RoboDK station: New Station (1).rdk

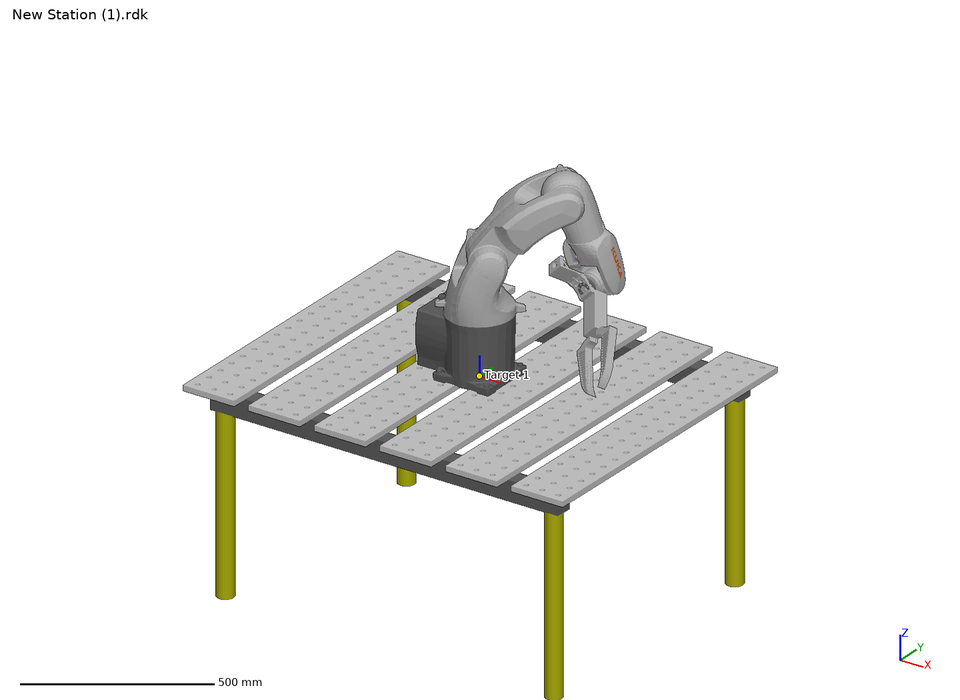
[picture v0: the station drawn from its stored meshes, robots at their saved joint values, targets as dots, program paths as lines]
Station New Station (1). Poses are relative to the parent item; angles as X-Y-Z fixed-axis rotations.
Station parameters (name, value as stored): DO_NAME, 1, IO_2, 0, IO_1, 1
  - object Table at (0, 1063.9, 0) mm, size 1193.8 x 965.2 x 609.6 mm, geometry from welding_table.sld
  - frame KUKA KR 3 R540 Base at (0, 1061.83, 0) mm
    - robot KUKA KR 3 R540: 6 axes, payload 3 kg, reach 541 mm, repeatability 0.02 mm, weight 26 kg
        modified DH rows (alpha deg, a mm, theta deg, d mm): 0, 0, 0, 345; -90, 20, 0, 0; 0, 260, -90, 0; -90, 20, 0, 260; 90, 0, 0, 0; -90, 0, 180, 75
        joint limits [-170, -170, -110, -175, -120, -350] to [170, 50, 155, 175, 120, 350]; home [0, -90, 90, 0, 0, 0]; saved at [-39.041, -39.658, 113.258, 52.118, 100.244, -32.123]
      - tool , TCP at (-200, -20, 130) mm, size 354.8 x 148.9 x 225.7 mm, geometry from .stl
    - target Target 1 (Cartesian target) at (0, 0, 0) mm, rotated rx -90 ry -45 rz 180 deg; joints [-93.946, 23.529, 82.573, -4.107, 73.937, -43.862] of KUKA KR 3 R540
  - Python program Смыкание и размыкание клешни (listed below)
  - program Раздвиг (4 instructions, listed below)
  - program Сдвиг (4 instructions, listed below)
  - program Prog8 (6 instructions, listed below)
  - Python program ts (listed below)
  - Python program tes (listed below)

--- Python program Смыкание и размыкание клешни ---
# Type help("robolink") or help("robodk") for more information
# Press F5 to run the script
# Note: you do not need to keep a copy of this file, your python script is saved with the station
from robolink import *    # API to communicate with RoboDK
from robodk import *      # basic matrix operations
RDK = Robolink()

# This file allows simulating the opening and closing of grippers.
# Two models of the gripper per robot are required: one opened and one closed.
# The opened model of the gripper should have the keyword "Opened"
# The closed model of the gripper should have the keyword "Closed"
# Simply place this file in the station and leave it running to
# make it work
program = RDK.AddProgram('program')
program.setDO('DO_NAME', 0)
program.setDO('DO_NAME', 1)
OPENED_KEYWORD = 'Opened'
CLOSED_KEYWORD = 'Closed'
UPDATE_FREQUENCY = 0.01

# Loop forever
print('Starting infinite loop to simulate open/close of tools')
while True:
    # First step: get a list of tool pairs (open, closed) per robot
    Tool_Pairs = []
    # get all the robot names (strings)
    all_robots = RDK.ItemList(ITEM_TYPE_ROBOT, True)
    for i in range(len(all_robots)):
        roboti = RDK.Item(all_robots[i])
        roboti_name = roboti.Name()
        # get the tools of each robot
        roboti_tools = roboti.Childs()
        opened = None
        closed = None
        # store the opened model and closed model of each gripper
        for t in range(len(roboti_tools)):
            tnamei = roboti_tools[t].Name()
            if not isinstance(opened,Item) and tnamei.count(OPENED_KEYWORD) > 0:
                opened = roboti_tools[t]
                print('Using %s from robot %s as gripper opened' % (tnamei, roboti_name))
            elif not isinstance(closed,Item) and tnamei.count(CLOSED_KEYWORD) > 0:
                closed = roboti_tools[t]
                print('Using %s from robot %s as gripper closed' % (tnamei, roboti_name))

            if isinstance(opened, Item) and isinstance(closed, Item):
                # Stop if we have an open state and a closed state per robot
                break;
        Tool_Pairs.append([opened, closed])

    # We may find as many pairs of tools as robots are available in the station
    nTool_Pairs = len(Tool_Pairs)
    while True:
        #try:
                # Iterate through all tool pairs and detect the presence of objects
            for i in range(nTool_Pairs):
                opened = Tool_Pairs[i][0]
                closed = Tool_Pairs[i][1]
                open_valid = isinstance(opened,Item)
                close_valid = isinstance(closed,Item)
                tool_is_open = True

                # Check if the tool holds one or more objects:
                if (open_valid and len(opened.Childs()) > 0) or (close_valid and len(closed.Childs()) > 0):
                    tool_is_open = False

                # Update the visibility of the tools
                if open_valid:
                    opened.setVisible(tool_is_open)
                if close_valid:
                    closed.setVisible(not tool_is_open)

            # Take a pause...
            pause(UPDATE_FREQUENCY)

                #except:
                     #print('An item was deleted. Remaking tool list')
                #break

--- program Раздвиг (robot KUKA KR 3 R540) ---
  Set IO_2=0
  Pause 1.0 s
  Set IO_1=1
  Pause 1.0 s

--- program Сдвиг (robot KUKA KR 3 R540) ---
  Set IO_2=1
  Pause 1.0 s
  Set IO_1=0
  Pause 1.0 s

--- program Prog8 (robot KUKA KR 3 R540) ---
  Call ts
  Call Сдвиг
  Call ts
  Call ts
  Call ts
  Call Раздвиг

--- Python program ts ---
import time
import serial
from robodk import*
from robolink import*
RDK = Robolink()
robot = RDK.Item("KUKA KR 3 R540")
target = RDK.Item("Target 1")

ser = serial.Serial('COM9', 9600)
time.sleep(2)
s = ser.readline()
a = str(s)[2:][:-5]
glist = list(a.split(" "))
x = int(glist[0])
y = int(glist[1])
z = int(glist[2])
x *= -1
z *= -1

approach = target.Pose()*transl(x, y, z)
robot.MoveJ(approach)

--- Python program tes ---
from robodk import*
from robolink import*
RDK = Robolink()
robot = RDK.Item("UR 10")
target = RDK.Item("Target 1")
x = 400
y = 0
z = 220
x *= -1
z *= -1
robot.setJoints([0, 0, 0, 0, 90, 180])
approach = target.Pose()*transl(x, y, z)
robot.MoveJ(approach)
